TYPE EL6910_ESTOP :
STRUCT
	
	diagnostics : EL6910_ESTOP_DIGNOSTICS;
	status	: EL6910_ESTOP_STATUS;	

END_STRUCT
END_TYPE

(* stored: Version 1.1.0.1, ProductVersion 3.1.4024.15
   DUT EL6910_ESTOP: Id {a638af62-71a3-456b-a53b-798b1a02c9e1} *)
